ABB RobotStudio station: sesion4.rsstn

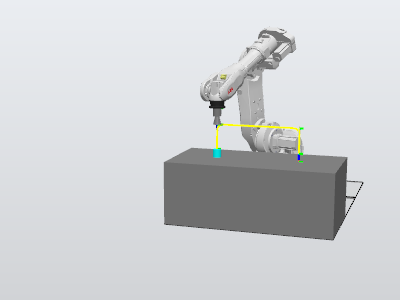
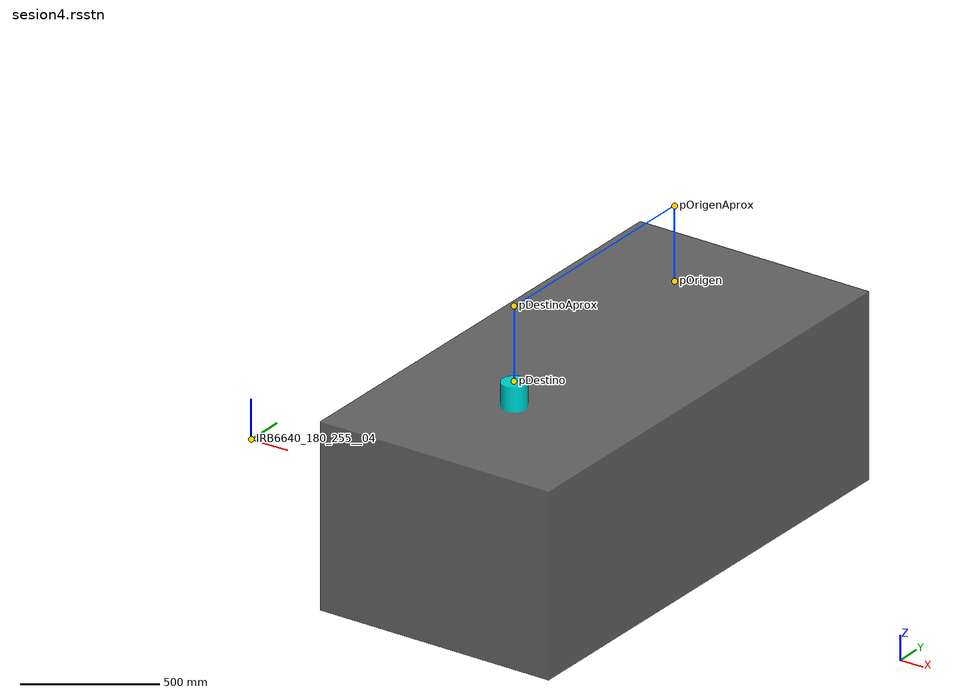
[picture v1: parts stored in the station drawn from their meshes, with robot base, taught points and paths (robot models come from the ABB library and are not in the file)]
Station sesion4 (saved by RobotStudio 24.1.10713.1)
Controller Controlador3
  mechanical unit ROB_1: IRB6640_180_255__04, 6 joints, base frame (0, 0, 0) mm
Layout (positions relative to the parent item):
  - Ventosa [mechanism] at (1500, -500, 1350) mm, rotated rx 180 ry 0 rz 180 deg
      TCP Ventosa at (0, 0, 200) mm
      links: PiezaVentosa
  - IRB6640_180_255__04 [mechanism, from %ABB.RobotStudio.Models.IRB6640%\IRB6640_180_255_G_04.rslib] at (0, 0, 0) mm; joint values [-0.3218, 0.1303, 0.301, 0, 1.1395, -0.3218] (rad or m)
  - Pieza_4 [part], size 1000 x 1000 x 750 mm
  - Pieza_5 [part], size 1000 x 1000 x 750 mm
  - Pieza_6 [part] at (0, -1000, 0) mm, size 100 x 99.8 x 100 mm
  - CI_VentosaVacuostato [smart component]
      signals: DO PiezaDetectada, DI ActivaVentosa, DO PiezaCogida
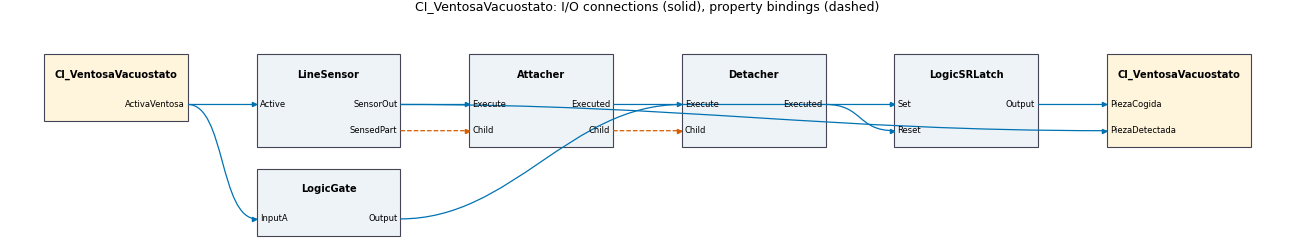
      connections:
        CI_VentosaVacuostato.ActivaVentosa -> LineSensor.Active
        LineSensor.SensorOut -> Attacher.Execute
        Attacher.Executed -> LogicSRLatch.Set
        LogicSRLatch.Output -> CI_VentosaVacuostato.PiezaCogida
        LineSensor.SensorOut -> CI_VentosaVacuostato.PiezaDetectada
        CI_VentosaVacuostato.ActivaVentosa -> LogicGate.InputA
        LogicGate.Output -> Detacher.Execute
        Detacher.Executed -> LogicSRLatch.Reset
        LineSensor.SensedPart => Attacher.Child
        Attacher.Child => Detacher.Child
    - LineSensor [smart component, from Components\LineSensor.rslib] at (1500, -500, 1150) mm, rotated rx 180 ry 0 rz 180 deg
        properties: Start=[0 0 -0.002]; End=[0 0 0.02]; Length=0.022; Radius=0.00210526315789474; Tag=(none); SensedPart=Pieza_6; SensedPoint=[1.50000012207031 -0.500000030517578 0.85]
      - _sensorPart_ [part], size 4.2 x 4.2 x 22 mm
    - LogicSRLatch [smart component, from Components\LogicSRLatch.rslib]
    - Attacher [smart component, from Components\Attacher.rslib]
        properties: Parent=Ventosa; Flange=0; Child=Pieza_6; Mount=false; Offset=[0 0 0]; Orientation=[0 0 0]
    - Detacher [smart component, from Components\Detacher.rslib]
        properties: Child=Pieza_6; KeepPosition=true
    - LogicGate [smart component, from Components\LogicGate.rslib]
        properties: Operator=NOT; Delay=0
Attachment: Ventosa is attached to IRB6640_180_255__04 / Link6
Attachment: LineSensor is attached to Ventosa / PiezaVentosa
Station logic (signal -> signal, property => property):
  CI_VentosaVacuostato.PiezaDetectada -> Controlador3.ED_PiezaDetectada
  Controlador3.SD_ActivaVentosa -> CI_VentosaVacuostato.ActivaVentosa
  CI_VentosaVacuostato.PiezaCogida -> Controlador3.ED_PiezaCogida
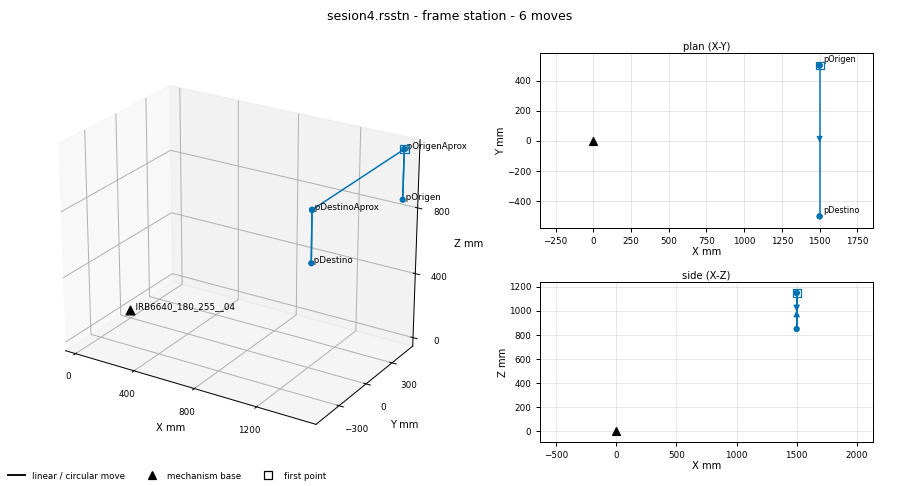
[picture p0: tool path of sesion4.rsstn in frame station, 6 of 6 moves have a stored position in this frame; points joined in program order, loops and branches not executed]
Targets, tools, work objects and paths stored in the station, written as RAPID:
! task T_ROB1
MODULE CalibData
  PERS tooldata Ventosa:=[TRUE,[[0,0,200],[1,0,0,0]],[1,[0,0,125],[1,0,0,0],0.002,0.002,0.0013]];
ENDMODULE

! task T_ROB1
MODULE Module1
  CONST robtarget pBaseOrigen:=[[1500,500,750],[0,0,1,0],[0,0,0,0],[9E+09,9E+09,9E+09,9E+09,9E+09,9E+09]];
  CONST robtarget pBaseDestino:=[[1500,-500,750],[0,0,1,0],[0,0,0,0],[9E+09,9E+09,9E+09,9E+09,9E+09,9E+09]];
  CONST robtarget pOrigen:=[[1500,500,850],[0,0,1,0],[0,0,0,0],[9E+09,9E+09,9E+09,9E+09,9E+09,9E+09]];
  CONST robtarget pDestino:=[[1500,-500,850],[0,0,1,0],[-1,0,-1,0],[9E+09,9E+09,9E+09,9E+09,9E+09,9E+09]];
  CONST robtarget pOrigenAprox:=[[1500,500,1150],[0,0,1,0],[0,0,0,0],[9E+09,9E+09,9E+09,9E+09,9E+09,9E+09]];
  CONST robtarget pDestinoAprox:=[[1500.000049807,-500.000011712,1150.000037959],[-0.000000035,0.000000015,1,0.000000012],[-1,-1,-1,0],[9E+09,9E+09,9E+09,9E+09,9E+09,9E+09]];
  PROC Path_10()
    MoveJ pOrigenAprox,v1000,z100,Ventosa\WObj:=wobj0;
    MoveL pOrigen,v400,fine,Ventosa\WObj:=wobj0;
    MoveL pOrigenAprox,v400,z100,Ventosa\WObj:=wobj0;
    MoveL pDestinoAprox,v2000,z100,Ventosa\WObj:=wobj0;
    MoveL pDestino,v400,fine,Ventosa\WObj:=wobj0;
    MoveL pDestinoAprox,v400,fine,Ventosa\WObj:=wobj0;
  ENDPROC
ENDMODULE

